(* Logix 5000 project; controller TORQUE Emulate 5570 rev 36.11; software revision 36.00 *)

TASK MainTask (continuous, watchdog 500 ms) : MainProgram, Emulation

MODULES
   Local : Emulate 5570 (ICP 2, rev 36.11)
       : 1756-IB16 (ICP 3, rev 3.1, Input RPI 20 ms)
       : vendor 1 type 7 code 16 (ICP 4, rev 3.1, Output RPI 20 ms)
       : 1756-IF8 (ICP 5, rev 1.1, Input RPI 100 ms)
END_MODULES

VAR_GLOBAL   (* controller tags *)
   AIN_1 : ALIAS FOR Local:5:I.Ch0Data;   // Channel 1, Torque Sensor No. 1
   AIN_2 : ALIAS FOR Local:5:I.Ch1Data;   // Channel 2, Torque Sensor No. 2
   AIN_3 : ALIAS FOR Local:5:I.Ch2Data;   // Channel 3, Torque Sensor No. 3
   AIN_4 : ALIAS FOR Local:5:I.Ch3Data;   // Channel 4, Torque Sensor No. 4
   DN_LS : ALIAS FOR Local:3:I.Data.0;   // Down Travel N.O. Limit Switch
   DN_SOL : ALIAS FOR Local:4:O.Data.0;   // Down Solenoid
   LOWER_LIMIT : DINT := 95;   // Lower Torque Setting
   MOTOR_1 : ALIAS FOR Local:4:O.Data.1;   // Nut Runner No. 1, Air Motor
   MOTOR_2 : ALIAS FOR Local:4:O.Data.2;   // Nut Runner No. 2, Air Motor
   MOTOR_3 : ALIAS FOR Local:4:O.Data.3;   // Nut Runner No. 3, Air Motor
   MOTOR_4 : ALIAS FOR Local:4:O.Data.4;   // Nut Runner No. 4, Air Motor
   START_NO_1 : ALIAS FOR Local:3:I.Data.14;   // START No. 1 Pushbutton
   START_NO_2 : ALIAS FOR Local:3:I.Data.15;   // START No. 2 Pushbutton
   TO_ERROR : ALIAS FOR Local:4:O.Data.10;   // Time Out Indicator
   UPPER_LIMIT : DINT := 100;   // Upper Torque Setting
END_VAR

PROGRAM Emulation   (* main routine Emulation *)
VAR
   emCROSS_THRD : BOOL;
   emDOWN_SOL_TRAVEL : TIMER := (PRE := 4000);
   emMOTOR1_ONS : BOOL;
   emMOTOR2_ONS : BOOL;
   emMOTOR3_ONS : BOOL;
   emMOTOR4_ONS : BOOL;
   emMOTOR_1_AIN : DINT := 76;
   emMOTOR_1_NO_TORQUE : BOOL := 1;
   emMOTOR_1_OFF_DWELL : TIMER := (PRE := 20);
   emMOTOR_1_ON_DWELL : TIMER := (PRE := 80);
   emMOTOR_2_AIN : DINT := 97;
   emMOTOR_2_ON_DWELL : TIMER := (PRE := 50);
   emMOTOR_3_AIN : DINT := 97;
   emMOTOR_3_ON_DWELL : TIMER := (PRE := 60);
   emMOTOR_4_AIN : DINT := 97;
   emMOTOR_4_CRS_DWELL : TIMER := (PRE := 20);
   emMOTOR_4_ON_DWELL : TIMER := (PRE := 20);
   emNO_TORQUE : BOOL := 1;
   emPART_TRACK : COUNTER := (PRE := 3, ACC := 3, CU := 1, DN := 1);
   emSET_POINT : DINT := 97;
END_VAR

ROUTINE Emulation   (* ladder *)
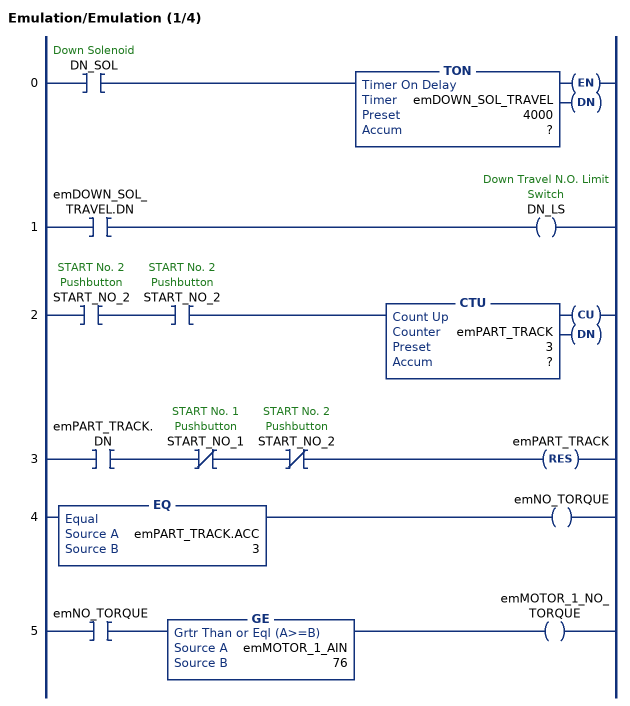
   0: XIC(DN_SOL)TON(emDOWN_SOL_TRAVEL,?,?);
   1: XIC(emDOWN_SOL_TRAVEL.DN)OTE(DN_LS);
   2: XIC(START_NO_2)XIC(START_NO_2)CTU(emPART_TRACK,?,?);
   3: XIC(emPART_TRACK.DN)XIO(START_NO_1)XIO(START_NO_2)RES(emPART_TRACK);
   4: EQ(emPART_TRACK.ACC,3)OTE(emNO_TORQUE);
   5: XIC(emNO_TORQUE)GE(emMOTOR_1_AIN,76)OTE(emMOTOR_1_NO_TORQUE);
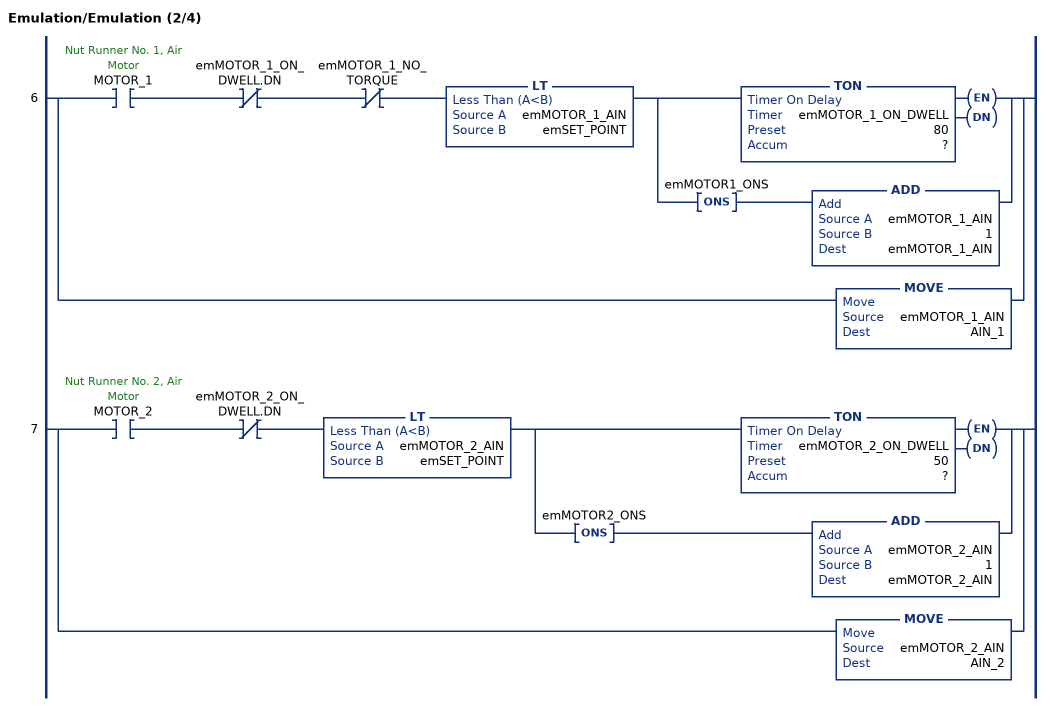
   6: [XIC(MOTOR_1) XIO(emMOTOR_1_ON_DWELL.DN) XIO(emMOTOR_1_NO_TORQUE) LT(emMOTOR_1_AIN,emSET_POINT) [TON(emMOTOR_1_ON_DWELL,?,?) ,ONS(emMOTOR1_ONS) ADD(emMOTOR_1_AIN,1,emMOTOR_1_AIN) ] ,MOVE(emMOTOR_1_AIN,AIN_1) ];
   7: [XIC(MOTOR_2) XIO(emMOTOR_2_ON_DWELL.DN) LT(emMOTOR_2_AIN,emSET_POINT) [TON(emMOTOR_2_ON_DWELL,?,?) ,ONS(emMOTOR2_ONS) ADD(emMOTOR_2_AIN,1,emMOTOR_2_AIN) ] ,MOVE(emMOTOR_2_AIN,AIN_2) ];
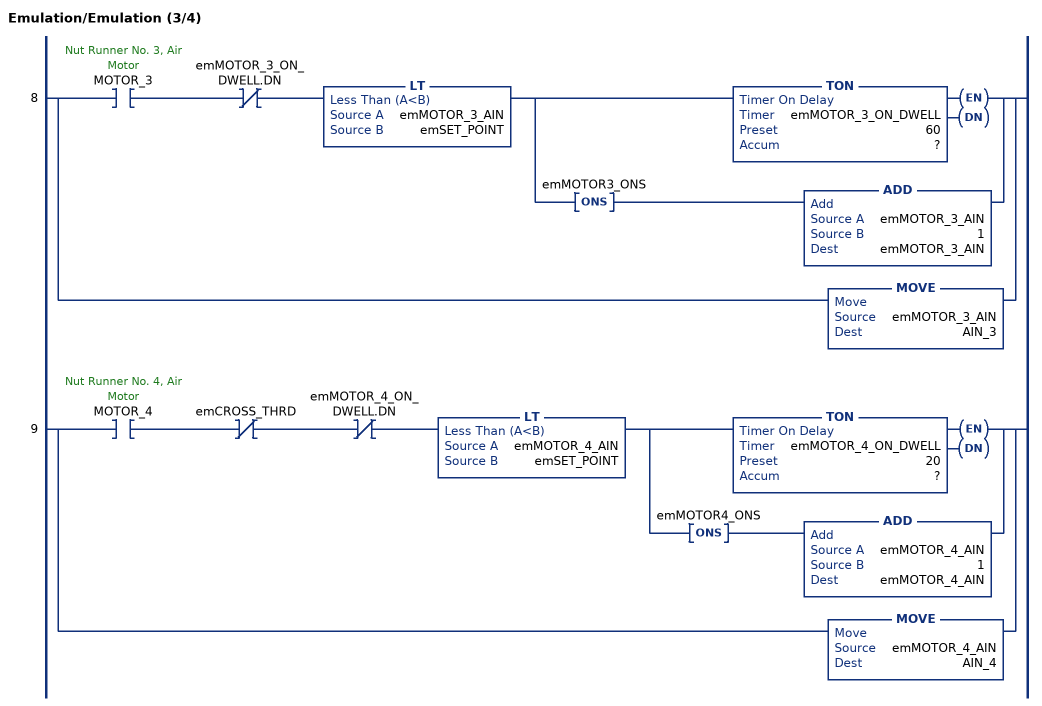
   8: [XIC(MOTOR_3) XIO(emMOTOR_3_ON_DWELL.DN) LT(emMOTOR_3_AIN,emSET_POINT) [TON(emMOTOR_3_ON_DWELL,?,?) ,ONS(emMOTOR3_ONS) ADD(emMOTOR_3_AIN,1,emMOTOR_3_AIN) ] ,MOVE(emMOTOR_3_AIN,AIN_3) ];
   9: [XIC(MOTOR_4) XIO(emCROSS_THRD) XIO(emMOTOR_4_ON_DWELL.DN) LT(emMOTOR_4_AIN,emSET_POINT) [TON(emMOTOR_4_ON_DWELL,?,?) ,ONS(emMOTOR4_ONS) ADD(emMOTOR_4_AIN,1,emMOTOR_4_AIN) ] ,MOVE(emMOTOR_4_AIN,AIN_4) ];
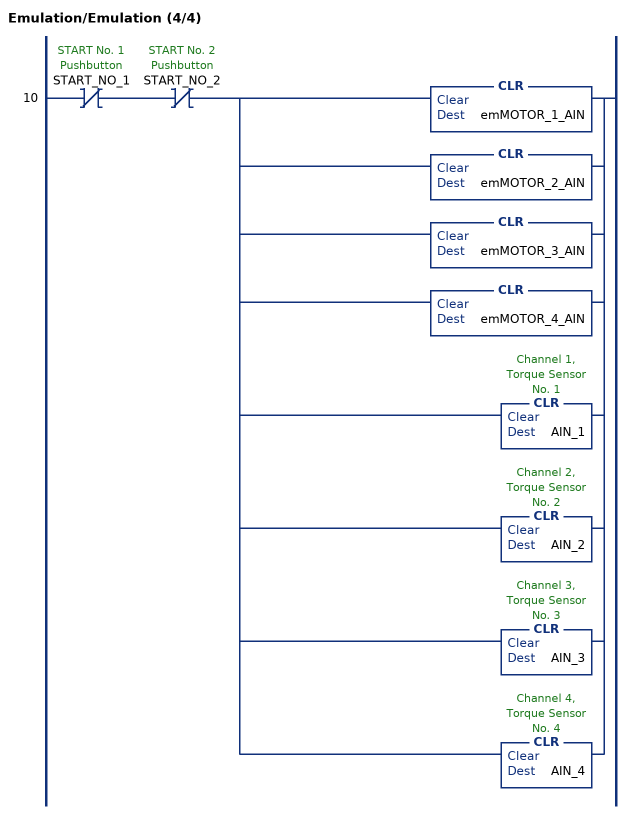
   10: XIO(START_NO_1)XIO(START_NO_2)[CLR(emMOTOR_1_AIN) ,CLR(emMOTOR_2_AIN) ,CLR(emMOTOR_3_AIN) ,CLR(emMOTOR_4_AIN) ,CLR(AIN_1) ,CLR(AIN_2) ,CLR(AIN_3) ,CLR(AIN_4) ];
END_ROUTINE
END_PROGRAM

PROGRAM MainProgram   (* main routine MainRoutine *)
VAR
   TO_DWELL : TIMER := (PRE := 20000, ACC := 20010, DN := 1);   // Time Out Dwell
        .DN   // Set Time Out Error (DN)
        .TT   // Time Out Elaspsing (TT) optional
        .EN   // Time Out Enabled (EN) Optional
   TORQUE_1_SET : BOOL;   // No. 1 Bolt Torque Set
   TORQUE_2_SET : BOOL := 1;   // No. 2 Bolt Torque Set
   TORQUE_3_SET : BOOL := 1;   // No. 3 Bolt Torque Set
   TORQUE_4_SET : BOOL := 1;   // No. 4 Bolt Torque Set
END_VAR

ROUTINE MainRoutine   (* ladder *)
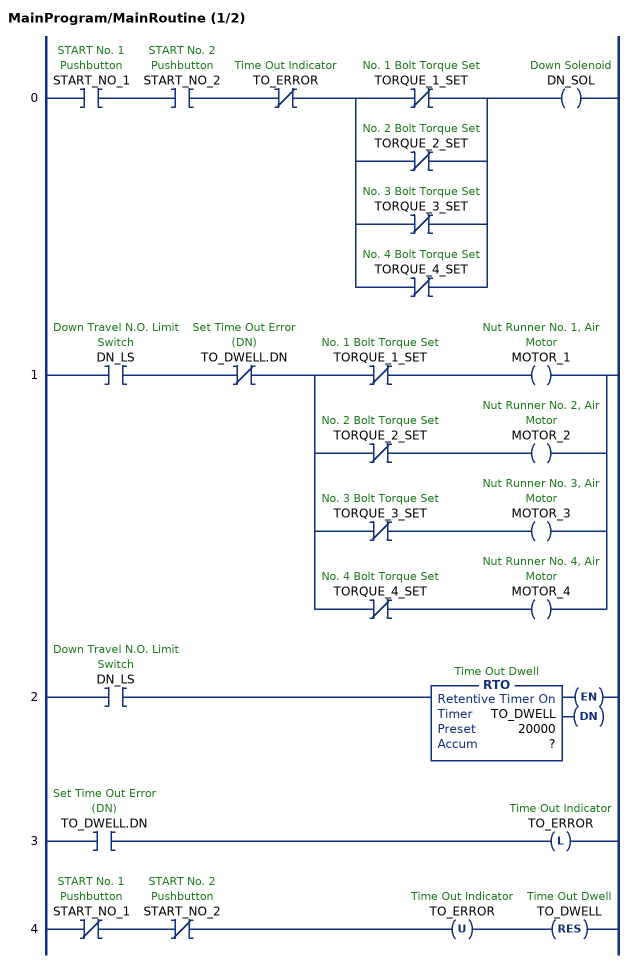
   0: XIC(START_NO_1)XIC(START_NO_2)XIO(TO_ERROR)[XIO(TORQUE_1_SET) ,XIO(TORQUE_2_SET) ,XIO(TORQUE_3_SET) ,XIO(TORQUE_4_SET) ]OTE(DN_SOL);
   1: XIC(DN_LS)XIO(TO_DWELL.DN)[XIO(TORQUE_1_SET) OTE(MOTOR_1) ,XIO(TORQUE_2_SET) OTE(MOTOR_2) ,XIO(TORQUE_3_SET) OTE(MOTOR_3) ,XIO(TORQUE_4_SET) OTE(MOTOR_4) ];
   2: XIC(DN_LS)RTO(TO_DWELL,?,?);
   3: XIC(TO_DWELL.DN)OTL(TO_ERROR);
   4: XIO(START_NO_1)XIO(START_NO_2)OTU(TO_ERROR)RES(TO_DWELL);
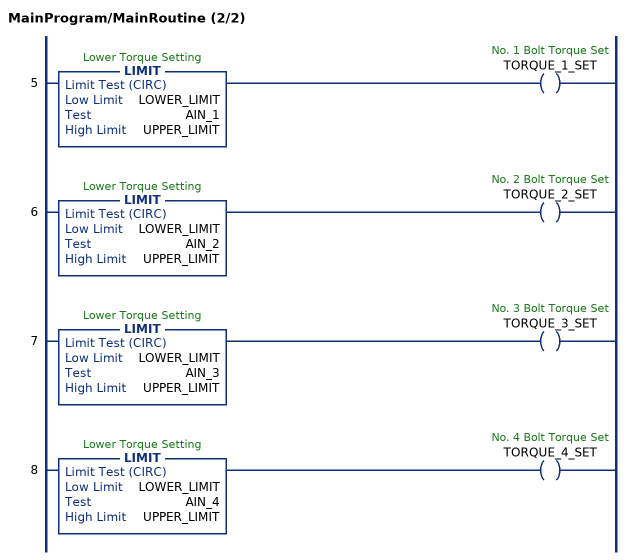
   5: LIMIT(LOWER_LIMIT,AIN_1,UPPER_LIMIT)OTE(TORQUE_1_SET);
   6: LIMIT(LOWER_LIMIT,AIN_2,UPPER_LIMIT)OTE(TORQUE_2_SET);
   7: LIMIT(LOWER_LIMIT,AIN_3,UPPER_LIMIT)OTE(TORQUE_3_SET);
   8: LIMIT(LOWER_LIMIT,AIN_4,UPPER_LIMIT)OTE(TORQUE_4_SET);
END_ROUTINE
END_PROGRAM
